FUNCTION WRITE_ANY_TIME : BOOL
VAR_INPUT
    ptr: POINTER TO TIME;
    val: TIME;
END_VAR

ptr^ := val;

END_FUNCTION

(* stored: Version 1.1.0.1, ProductVersion 3.1.4022.9
   POU WRITE_ANY_TIME: Id {fe63062b-7425-40a7-aecc-017a028de247}, SpecialFunc None *)
